// TIA Portal V20 export
DATA_BLOCK "DataToSafety"   // DB120
// stored: Access Published, InstanceOfName Safety.typeDataToSafety, InstanceOfType UDT, Namespace Safety
"Safety.typeDataToSafety"
   // VAR
   //    ackSafetyFromHmi : Int;
   //    ackSafetyGlobal : Bool;
   //    ackFromUnit1 : Bool;
   //    ackSafetyFromMobileHMI : Bool;
   //    resetSafetyFromMobileHMI : Bool;
   //    connectionBoxID_1 : Int;
   //    connectionBoxID_2 : Int;
   //    MobilePanelConnected : Bool;
   //    MobilePanelPermissions : Bool;
   //    DeselectBA10 : Bool;
   //    DeselectBA15 : Bool;
   //    DeselectBA40 : Bool;
   //    DeselectBA60 : Bool;
   //    PowerOnCommand : Bool;
   //    InitializeEnable : Bool;   // Main OP HOME
   //    BA060STOP : Bool;
   //    SepaGripperAxisXmoveToBa60 : Bool;
   //    unitMode : "Safety.typeUnitMode";
   //    BA060Mode : "Safety.typeUnitMode";
   //    unitState : "Safety.typeUnitStatus";
   //    winderUsed : "Safety.typeWinderUseMode";
   //    StackDoor1 : "Safety.typeFdoorCommands";
   //    StackDoor2 : "Safety.typeFdoorCommands";
   //    StackDoor6 : "Safety.typeFdoorCommands";
   //    StackDoor7 : "Safety.typeFdoorCommands";
   //    scrapBox1Monitoring : "Safety.typeScrapBoxMonitoring";
   //    scrapBox2Monitoring : "Safety.typeScrapBoxMonitoring";
   //    hotWireCutterCmds : "Safety.typeHotWireCutter";
   //    clock : "Safety.typeGlobalClockMem";
   //    BrakeTest { S7_SetPoint := 'True'} : "Safety.typeBrakeTest";
   // END_VAR
BEGIN
END_DATA_BLOCK
